PROGRAM MAIN
VAR
	Machine : Machine('Machine');
END_VAR

IF NOT Machine.Initialized THEN
	Machine.Initialize();
	RETURN;
END_IF

Machine.CyclicLogic();

END_PROGRAM

(* stored: Version 1.1.0.1, ProductVersion 3.1.4026.18
   POU MAIN: Id {64551e79-26ad-474c-b7db-26dbd776d24f}, SpecialFunc None *)
